// TIA Portal V18 export
DATA_BLOCK "Auxiliary_variables"   // DB17
{ S7_Optimized_Access := 'TRUE' }
VERSION : 0.1
// stored: AutoNumber true, DBAccessibleFromOPCUA true, IsOnlyStoredInLoadMemory false, IsRetainMemResEnabled false, IsWriteProtectedInAS false, MemoryReserve 100
   VAR
      GlobalEnableAxis : Bool;   // Variable enables Enable_machine [FC5]
      DisableAxis : Bool;   // Variable enables Stop_machine_sequence [FC4]
      StartFunction : Bool;   // Variable enables Function_sequence [FC6]
      ESTOP : Bool;   // Variable enables Emergancy_stop_sequence [FC3]
      ResetErrors : Bool;   // Variable enables Reset_error_sequence [FB14]
      Position_range_Z2 : DInt;   // Check if position is in the range Z2
      Mov_permission_Z2_Absolute : Bool;   // Permission to move Z2 (Input Axis_Mov Z2)
      Mov_permission_Z2_Relative : Bool;
      Stop_Z2_Out : Bool;   // Stop Z2 movement (Output for Axis_Mov Z2 block)
      Reset_command_Z2 : Bool;   // Reset Mov_mode / Mode_mode = 0 / Input for BOOL_DEMUX and Output for Axis_Mov Z2 Block
      Reset_error_jump_Z2 : Bool;   // Using in order to eliminate double write
      Position_range_X : DInt;   // Check if position is in the range X
      Mov_permission_X_Absolute : Bool;   // Permission to move Z2 (Input Axis_Mov X)
      Mov_permission_X_Relative : Bool;
      Stop_X_Out : Bool;   // Stop X movement (Output for Axis_Mov X block)
      Reset_command_X : Bool;   // Reset Mov_mode / Mode_mode = 0 / Input for BOOL_DEMUX and Output for Axis_Mov X Block
      Reset_error_jump_X : Bool;   // Using in order to eliminate double write
      Reset_command_Y : Bool;   // Reset Mov_mode / Mode_mode = 0 / Input for BOOL_DEMUX and Output for Axis_Mov Y Block
      Reset_error_jump_Y : Bool;   // Using in order to eliminate double write
      Stop_Y_Out : Bool;   // Stop Y movement (Output for Axis_Mov Y block)
      Mov_permission_Y_Absolute : Bool;   // Permission to move Y (Input Axis_Mov Y)
      Mov_permission_Y_Relative : Bool;
      Position_range_Y : DInt;   // Check if position is in the range Y
      Position_range_Z1 : DInt;   // Check if position is in the range Z1
      Mov_permission_Z1_Absolute : Bool;   // Permission to move Z1 (Input Axis_Mov Z1)
      Mov_permission_Z1_Relative : Bool;
      Stop_Z1_Out : Bool;   // Stop Z1 movement (Output for Axis_Mov Z1 block)
      Reset_command_Z1 : Bool;   // Reset Mov_mode / Mode_mode = 0 / Input for BOOL_DEMUX and Output for Axis_Mov Z1 Block
      Reset_error_jump_Z1 : Bool;   // Using in order to eliminate double write
      Stop_all_axis_command : Bool;   // Execute via Step6 ( in Main) / Stop all axis
      Mov_mode_reset_ALL_Axis : Bool;   // Reset Mov_mode after stopping all axis
      JogPosBTN_Z1_RisingEdge : Bool;   // Auxiliary variable used to execute JogPos Button
      JogNegBTN_Z1_RisingEdge : Bool;   // Auxiliary variable used to execute JogNeg Button
      JogPosBTN_Z1_FallingEdge : Bool;   // Auxiliary variable used to execute JogPos Button
      JogNegBTN_Z1_FallingEdge : Bool;   // Auxiliary variable used to execute JogNeg Button
      JogPosBTN_Z2_RisingEdge : Bool;   // Auxiliary variable used to execute JogPos Button
      JogNegBTN_Z2_RisingEdge : Bool;   // Auxiliary variable used to execute JogNeg Button
      JogPosBTN_Z2_FallingEdge : Bool;   // Auxiliary variable used to execute JogPos Button
      JogNegBTN_Z2_FallingEdge : Bool;   // Auxiliary variable used to execute JogNeg Button
      Heater_Start : Bool;   // Variable used to activate the heater during the spreading sequence
      PID_PWM_Output : Bool;   // PID Compact block -> Output
      CMD_Y_EM : Bool;
      CMD_X_EM : Bool;
      CMD_Z1_EM : Bool;
      CMD_Z2_EM : Bool;
      RelativeZ1 : Bool;
   END_VAR
BEGIN
END_DATA_BLOCK
